TYPE ST_ItemLogBuffer :
STRUCT
	aBufferData	:	ARRAY [0..999] OF ST_Item;	// Data stored in the buffer, 100 elements
	nInPointer	:	UDINT;							// Pointer for data put into the buffer
END_STRUCT
END_TYPE

(* stored: Version 1.1.0.1, ProductVersion 3.1.4024.6
   DUT ST_ItemLogBuffer: Id {e3356e34-585a-4f77-8b1f-db0d645cc59d} *)
